Omron CX-Programmer project NewProject (CX-Programmer 9.75)

# PLC NewPLC1: CP2E-N N

## Global symbols (name address type ; comment)
0.00 BOOL  ; PROXY STOP KONVEYOR
0.01 BOOL  ; PROXY BOWL DISPENSER
0.02 BOOL  ; START BUTTON
100.00 BOOL  ; MOTOR BOWL DISPENSER
100.01 BOOL  ; MOTOR KONVEYOR
100.02 BOOL  ; MOTOR KONVEYOR
100.06 BOOL  ; MOTOR LINEAR ACTUATOR
200.00 BOOL  ; RELAY START
200.01 BOOL  ; RELAY START KONVEYOR
200.02 BOOL  ; RELAY ACTUATOR
200.03 BOOL  ; MOTOR BOWL
200.04 BOOL  ; RESET COUNTER
C0 CHANNEL  ; COMPILE MOTOR BOWL
T000 BOOL  ; TIMER ACTUATOR
T001 BOOL  ; TIMER START KONVEYOR
T002 BOOL  ; TIMER START KONVEYOR AFTER BOWL
T003 BOOL  ; START BOWL

## Program NewProgram1 (cyclic task 0)

### Section Section1

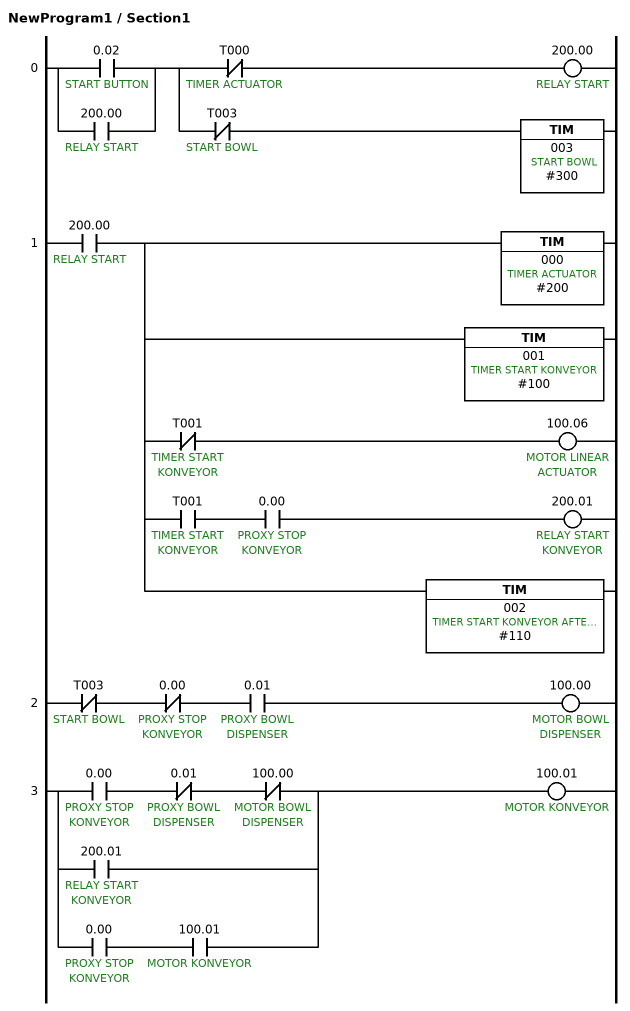
; rung 0
LD 0.02  ; START BUTTON
OR 200.00  ; RELAY START
OUT TR0
ANDNOT T000  ; TIMER ACTUATOR
OUT 200.00  ; RELAY START
LD TR0
ANDNOT T003  ; START BOWL
TIM 003 #300  ; START BOWL
; rung 1
LD 200.00  ; RELAY START
OUT TR0
TIM 000 #200  ; TIMER ACTUATOR
TIM 001 #100  ; TIMER START KONVEYOR
ANDNOT T001  ; TIMER START KONVEYOR
OUT 100.06  ; MOTOR LINEAR ACTUATOR
LD TR0
AND T001  ; TIMER START KONVEYOR
AND 0.00  ; PROXY STOP KONVEYOR
OUT 200.01  ; RELAY START KONVEYOR
LD TR0
TIM 002 #110  ; TIMER START KONVEYOR AFTER BOWL
; rung 2
LDNOT T003  ; START BOWL
ANDNOT 0.00  ; PROXY STOP KONVEYOR
AND 0.01  ; PROXY BOWL DISPENSER
OUT 100.00  ; MOTOR BOWL DISPENSER
; rung 3
LD 0.00  ; PROXY STOP KONVEYOR
ANDNOT 0.01  ; PROXY BOWL DISPENSER
ANDNOT 100.00  ; MOTOR BOWL DISPENSER
OR 200.01  ; RELAY START KONVEYOR
LD 0.00  ; PROXY STOP KONVEYOR
AND 100.01  ; MOTOR KONVEYOR
ORLD
OUT 100.01  ; MOTOR KONVEYOR

### Section END
; rung 0
END(001)